// CheckLRangeUnsigned checks subrange types of the type LWORD, ULINT.
// The purpose of this monitoring function is to deal with range bound violations as appropriate.
// Implicitly generated code : DO NOT EDIT
FUNCTION CheckLRangeUnsigned : ULINT
VAR_INPUT
	value, lower, upper: ULINT;
END_VAR

// Implicitly generated code : Only an Implementation suggestion
{noflow}
IF (value < lower) THEN
	CheckLRangeUnsigned := lower;
	GVL_TwinCatChecks.CheckRange_ULINT_TooLow := GVL_TwinCatChecks.CheckRange_ULINT_TooLow + 1;
ELSIF(value > upper) THEN
	CheckLRangeUnsigned := upper;
	GVL_TwinCatChecks.CheckRange_ULINT_TooHigh := GVL_TwinCatChecks.CheckRange_ULINT_TooHigh + 1;
ELSE
	CheckLRangeUnsigned := value;
END_IF
{flow}

END_FUNCTION

(* stored: Version 1.1.0.1, ProductVersion 3.1.4024.10
   POU CheckLRangeUnsigned: Id {70c7f2c4-5290-4802-9686-5c71ee93d2f1}, SpecialFunc CheckLRangeUnsigned *)
